{attribute 'linkalways'} 
{attribute 'no_explicit_call' := 'This FB is a CLASS and must be accessed using methods or properties'}
{attribute 'enable_dynamic_creation'}
FUNCTION_BLOCK RegisteredRpcApis
VAR
	registeredRpcApis : Queue;
	_hasRegisteredRpcApis : BOOL;
	enumerator : I_ForwardEnumerator;
END_VAR

METHOD PRIVATE CreateEnumerator
VAR_INPUT
END_VAR
IF enumerator <> 0 THEN
	enumerator.Dispose();
END_IF

enumerator := registeredRpcApis.GetEnumerator();
END_METHOD

METHOD PUBLIC CyclicCall
VAR
	rpcApi : I_RpcApi;
END_VAR
IF NOT HasRegisteredRpcApis THEN
	RETURN;
END_IF

enumerator.Reset();

WHILE enumerator.MoveNext() DO
	IF enumerator.TryGet(rpcApi) THEN
		rpcApi.CyclicCall();
	END_IF;
END_WHILE
END_METHOD

METHOD FB_exit : BOOL
VAR_INPUT
	bInCopyCode : BOOL; // if TRUE, the exit method is called for exiting an instance that is copied afterwards (online change).
END_VAR
IF bInCopyCode THEN
	RETURN;
END_IF

IF enumerator <> 0 THEN
	enumerator.Dispose();
END_IF
END_METHOD

PROPERTY PUBLIC HasRegisteredRpcApis : BOOL
GET
HasRegisteredRpcApis := enumerator <> 0;
END_GET
END_PROPERTY

METHOD PUBLIC RegisterRpcApi
VAR_INPUT
	RpcApi : I_RpcApi;
END_VAR
registeredRpcApis.Enqueue(RpcApi);
CreateEnumerator();
END_METHOD

END_FUNCTION_BLOCK

(* stored: Version 1.1.0.1, ProductVersion 3.1.4024.12
   POU RegisteredRpcApis: Id {da469a70-bfcd-4b8c-ae16-6c035db07b94}, SpecialFunc None
   Folder Destructor: Id {a58e1318-3e30-40eb-b3c6-32973c1a4711}
   Folder Private: Id {1114c840-a5e6-4269-9db3-0a90b4e5f6bb}
   Method CreateEnumerator: Id {8ce64f94-58ed-4311-8f4c-9677482592cf}
   Method CyclicCall: Id {98ddba6a-4b14-44d8-a8c4-1d829b26b1b4}
   Method FB_exit: Id {05c4b2ef-3d25-4b8b-8745-e773efee3135}
   Property HasRegisteredRpcApis: Id {d1c712f4-7a84-4041-8c80-2e1002825a37}
   Get Get: Id {d56f3e1b-d15c-44a7-a522-68c720b88e83}
   Method RegisterRpcApi: Id {8a13a021-83ba-43d6-acb1-9bc400d1a212} *)
